(* PLC project Unnamed, Unknown Unnamed 1 *)
(* stored: creationDateTime 2023-04-26T09:18:19, modificationDateTime 2023-04-27T11:20:28 *)

PROGRAM OPLC_SORTBYMOD
  VAR
    ATENTRY : BOOL;
    ATBACK : BOOL;
    LOWBOX : BOOL;
    HIGHBOX : BOOL;
    TURNTABLEENTRY : BOOL;
    LOADPOS : BOOL;
    UNLOADPOS : BOOL;
    ATFRONT : BOOL;
    RIGHTENT : BOOL;
    LEFTENT : BOOL;
    RIGHTEXIT : BOOL;
    LEFTEXIT : BOOL;
    START : BOOL;
    RESET : BOOL;
    STOP : BOOL;
    EMERGENCY : BOOL;
    MACH_ON : BOOL;
    MACH_OFF : BOOL;
    FEEDERCONV : BOOL;
    ENTRYCONV : BOOL;
    LOAD : BOOL;
    UNLOAD : BOOL;
    TURN : BOOL;
    LEFTCONV : BOOL;
    RIGHTCONV : BOOL;
    GREENIND : BOOL;
    YELLOWIND : BOOL;
    REDIND : BOOL;
    LSTART : BOOL;
    LRESET : BOOL;
    LSTOP : BOOL;
    CONT : BOOL;
    CONTINUERIGHT : BOOL;
    CONTINUELEFT : BOOL;
    TOF0 : TOF;
    ET : TIME;
    CTU0 : CTU;
    PV : WORD;
    CV : WORD;
    MEMOLEFT : BOOL;
    MEMORIGHT : BOOL;
    UNTURN : BOOL;
    SR0 : SR;
    SR1 : SR;
    TOF1 : TOF;
    TOF2 : TOF;
  END_VAR
  VAR  (* added by the conversion: wires and edge detectors of the diagram *)
    R_TRIG1 : R_TRIG;
  END_VAR

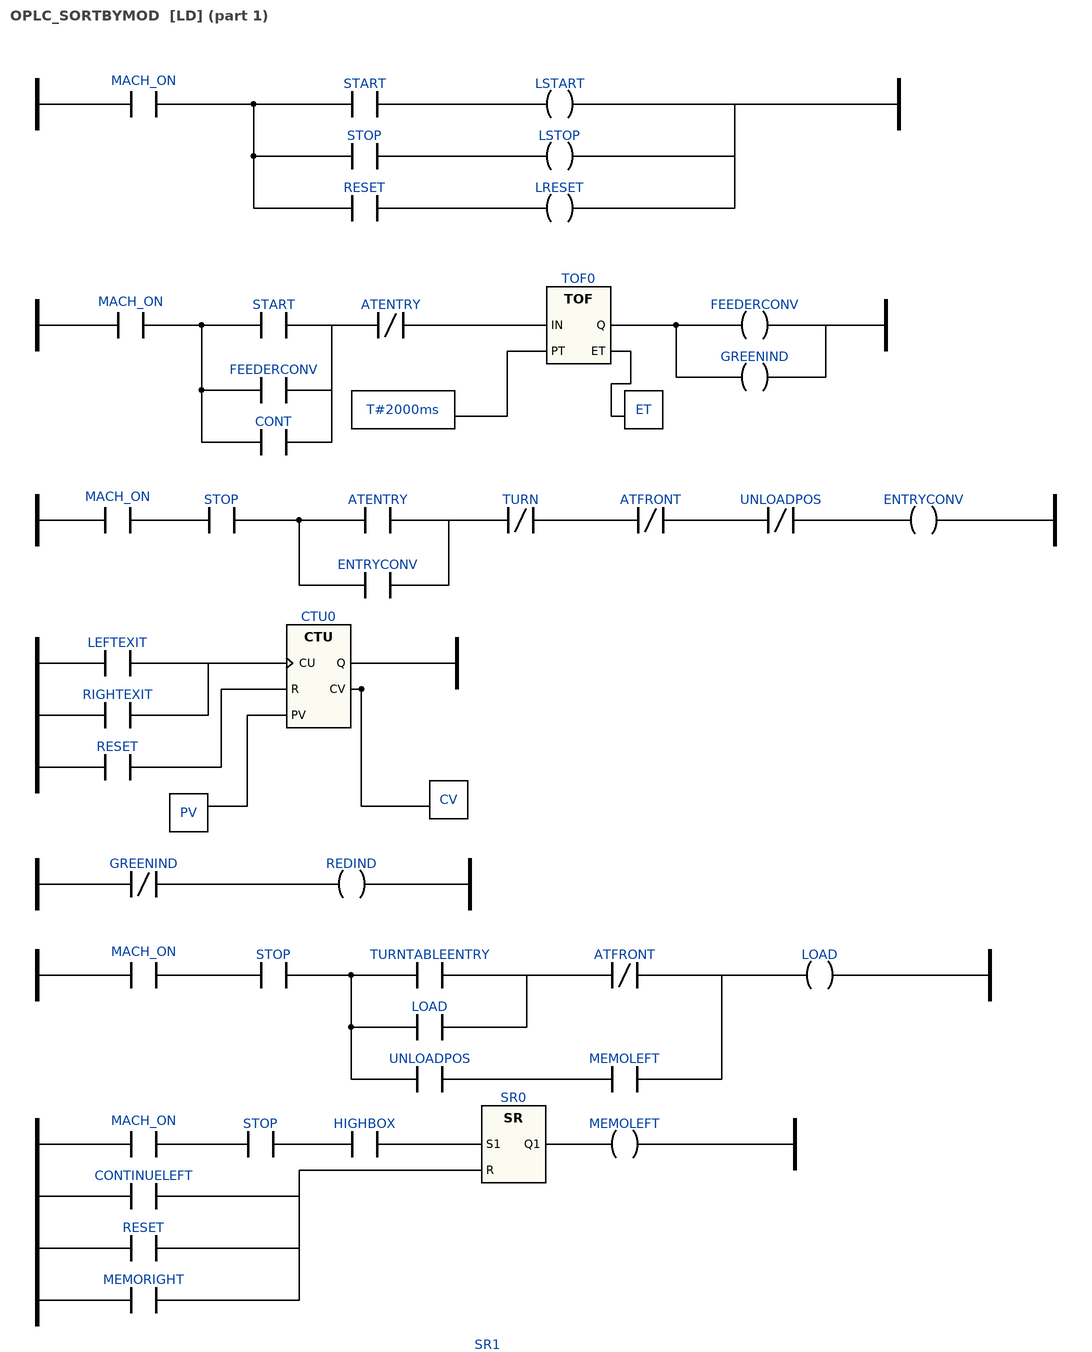
(* LD diagram, written out as Structured Text *)
LSTART := MACH_ON AND START;
LSTOP := MACH_ON AND STOP;
LRESET := MACH_ON AND RESET;
TOF0(IN := MACH_ON AND (START OR FEEDERCONV OR CONT) AND NOT ATENTRY, PT := T#2000ms);
FEEDERCONV := TOF0.Q;
GREENIND := TOF0.Q;
ET := TOF0.ET;
ENTRYCONV := MACH_ON AND STOP AND (ENTRYCONV OR ATENTRY) AND NOT TURN AND NOT ATFRONT AND NOT UNLOADPOS;
R_TRIG1(CLK := LEFTEXIT OR RIGHTEXIT);
CTU0(CU := R_TRIG1.Q, R := RESET, PV := PV);
CV := CTU0.CV;
REDIND := NOT GREENIND;
LOAD := MACH_ON AND STOP AND ((TURNTABLEENTRY OR LOAD) AND NOT ATFRONT OR UNLOADPOS AND MEMOLEFT);
SR0(S1 := MACH_ON AND STOP AND HIGHBOX, R := CONTINUELEFT OR RESET OR MEMORIGHT);
MEMOLEFT := SR0.Q1;
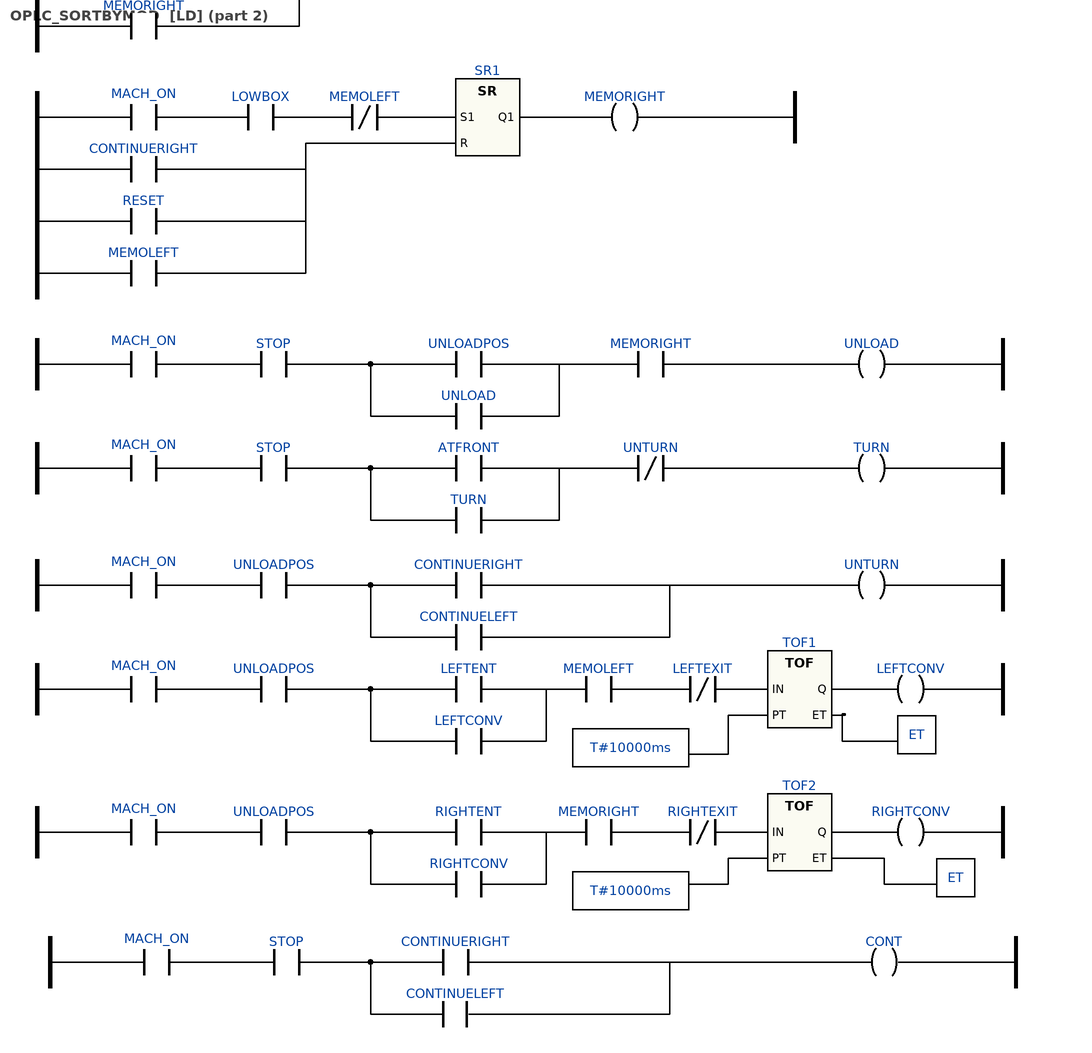
SR1(S1 := MACH_ON AND LOWBOX AND NOT MEMOLEFT, R := CONTINUERIGHT OR RESET OR MEMOLEFT);
MEMORIGHT := SR1.Q1;
UNLOAD := MACH_ON AND STOP AND (UNLOAD OR UNLOADPOS) AND MEMORIGHT;
TURN := MACH_ON AND STOP AND (TURN OR ATFRONT) AND NOT UNTURN;
UNTURN := MACH_ON AND UNLOADPOS AND (CONTINUERIGHT OR CONTINUELEFT);
TOF1(IN := MACH_ON AND UNLOADPOS AND (LEFTENT OR LEFTCONV) AND MEMOLEFT AND NOT LEFTEXIT, PT := T#10000ms);
LEFTCONV := TOF1.Q;
ET := TOF1.ET;
TOF2(IN := MACH_ON AND UNLOADPOS AND (RIGHTENT OR RIGHTCONV) AND MEMORIGHT AND NOT RIGHTEXIT, PT := T#10000ms);
RIGHTCONV := TOF2.Q;
ET := TOF2.ET;
CONT := MACH_ON AND STOP AND (CONTINUERIGHT OR CONTINUELEFT);
END_PROGRAM

CONFIGURATION Config0
  RESOURCE Res0 ON PLC
    TASK task0(INTERVAL := T#20ms, PRIORITY := 0);
    PROGRAM instance0 WITH task0 : OPLC_SORTBYMOD;
  END_RESOURCE
END_CONFIGURATION
